// TIA Portal V16 export
// export: Created 2023-03-29T11:04:37.7582368Z, ExportSetting WithDefaults, DisplayName Totally Integrated Automation Portal, DisplayVersion V16 Update 6, DisplayName TIA Portal Version Control Interface, DisplayVersion V16 Update 2, DisplayName TIA Portal Openness, DisplayVersion V16 Update 6, DisplayName STEP 7 Professional, DisplayVersion V16 Update 6, DisplayName STEP 7 Safety, DisplayVersion V16, DisplayName WinCC Advanced, DisplayVersion V16 Update 6
DATA_BLOCK "dbHold_RRG"   // DB57
TITLE = Instancja danych serwera TCP
{ S7_Optimized_Access := 'FALSE' }
AUTHOR : rtecmer
VERSION : 0.1
// Instancja dla serwera Modbus TCP. Dane udostępniane i wpisywanedla PLC Zasuwy
// stored: AutoNumber true, DBAccessibleFromOPCUA true, IsOnlyStoredInLoadMemory false, IsWriteProtectedInAS false
   VAR
      actB5_bar_magistrala : Real;   // 4001-4002 Pomiar ciśnienia magistrala - dosilanie
      act_poziom_ZB1 : Real;   // 4003-4004 Pomiar poziom w zbiorniku
      act_poziom_ZB2 : Real;   // 4005-4006 Pomiar poziom w zbiorniku
      act_poziom_ZB3 : Real;   // 4007-4008 Pomiar poziom w zbiorniku
      act_poziom_ZB4 : Real;   // 4009-4010 Pomiar poziom w zbiorniku
      act_przepływ_VF_Q2 : Real;   // 4011-4012 Aktualny przepływ VF
      "act_przepływ-VR_Q2" : Real;   // 4013-4014 Aktualny przepływ VR wsteczny
      sum_przepływ_Q2 : Real;   // 4015-4016
      status_Z1 : Word;   // 4017
      status_Z2 : Word;   // 4018
      status_Z3 : Word;   // 4019
      status_Z4 : Word;   // 4020
      status_Z5 : Word;   // 4021
      status_Z6 : Word;   // 4022
      status_Z7 : Word;   // 4023
      status_Z8 : Word;   // 4024
      status_Z9 : Word;   // 4025
      status_Z10 : Word;   // 4026
      status_przepływomierz_Q2 : Word;   // 4027 status przepływomierza DN500
      act_położenie_Z10 : Word;   // 4028 Położenie zasuwy Z10 [%]
      komunikacja_PLC : Word;   // 4029 Kontrola komunikacji PLC1 - PLC2 wartość 0 wysyłane do PLC1
      set_poziom_napełniania : Real;   // 4030 - 4031 wartość zadana poziomu napełniania
      set_poziom_opróżniania : Real := 30.0;   // 4032 - 4033 wartość zadana poziomu opróżniania
      set_res_bity_sterowania_napęami_1 : Word;   // 4034 bity sterowania napędami
      set_res_bity_sterowania_napęami_2 : Word;   // 4035 bity sterowania napędami
      set_res_bity_tryb_napędów_1 : Word;   // 4036 bity sterowania przełączaniem trybów pracy
      set_res_bity_tryb_napędów_2 : Word;   // 4037 bity sterowania przełączaniem trybów pracy
      reset_alarm_napędów : Word;   // 4038 bity kasowania alarmów napędów
      set_strategia_sterowania : Word;   // 4039 (Bit 53.0 - Wyłączony), (Bit 53.1 - Dosilanie), (Bit 53.2 - Przetłączanie), (Bit 53.3 - Automat), (Bit 53.4 - Ręczne )
      set_sterowanie_cyklem : Word;   // 4040 (Bit 55.0 - Cykl wyłączony (Bit 55.1 - Cykl dobowy), (Bit 55.2 - Cykl tygodniowy), (Bit 55.3 - Cykl ręczny)
      set_położenie_Z10 : Word;   // 4041Położenie zasuwy Z10 [%]
      komunikacjaPLC : Word;   // 4042 kontrola komunikacji wysyłanie -> 0
      start_napełnianie : DTL := DTL#1970-01-01-23:55:00;   // 4043
      Stop_napełnianie : DTL := DTL#1970-01-01-16:00:00;
      Start_przetłaczanie_1 : DTL := DTL#1970-01-01-18:00:00;
      Stop_przetłaczanie_1 : DTL := DTL#1970-01-01-23:40:00;
      Start_dosilanie_1 : DTL := DTL#1970-01-01-18:00:00;
      Stop_dosilanie_1 : DTL := DTL#1970-01-01-23:40:00;
      Sending : Struct
         act_położenie_Z10 : Word := 40;   // Położenie zasuwy Z11 [%]
         set_poziom_napełniania : Real := 550.0;   // wartość zadana poziomu napełniania
         set_poziom_opróżniania : Real := 30.0;   // wartość zadana poziomu opróżniania
         set_res_bity_sterowania_napęami_1 : Word;   // bity sterowania napędami
         set_res_bity_sterowania_napęami_2 : Word;   // bity sterowania napędami
         set_res_bity_tryb_napędów_1 : Word;   // bity sterowania przełączaniem trybów pracy
         set_res_bity_tryb_napędów_2 : Word;   // bity sterowania przełączaniem trybów pracy
         rez_alarm_napędów : Word;   // bity kasowania alarmów napędów
         set_strategia_sterowania : Word;   // (Bit 53.0 - Wyłączony), (Bit 53.1 - Dosilanie), (Bit 53.2 - Przetłączanie), (Bit 53.3 - Automat), (Bit 53.4 - Ręczne )
         set_sterowanie_cyklem : Word;   // (Bit 55.0 - Cykl wyłączony (Bit 55.1 - Cykl dobowy), (Bit 55.2 - Cykl tygodniowy), (Bit 55.3 - Cykl ręczny)
         set_położenie_Z10 : Word;   // zadane położenie procentowe Z10
         komunikacjaPLC : Word;   // kontrola komunikacji wysyłanie -> 0
         set_magistrala_alarm_min_bar : Real := 6.5;   // wartość alarmowa awaria zasilania na magistrali B5
      END_STRUCT;
      SendingTimes : Struct
         start_napełnianie : DTL := DTL#1970-01-01-23:55:00;
         Stop_napełnianie : DTL := DTL#1970-01-01-16:00:00;
         Start_przetłaczanie_1 : DTL := DTL#1970-01-01-18:00:00;
         Stop_przetłaczanie_1 : DTL := DTL#1970-01-01-23:40:00;
         Start_dosilanie_1 : DTL := DTL#1970-01-01-18:00:00;
         Stop_dosilanie_1 : DTL := DTL#1970-01-01-23:40:00;
      END_STRUCT;
   END_VAR
BEGIN
END_DATA_BLOCK
